{attribute 'linkalways'} 
{attribute 'no_explicit_call' := 'This FB is a CLASS and must be accessed using methods or properties'}
{attribute 'enable_dynamic_creation'}
FUNCTION_BLOCK _UDINT EXTENDS NumericDatatypeBase
VAR
	localData : UDINT;
	activeData : REFERENCE TO UDINT REF= localData;
END_VAR

PROPERTY PUBLIC Address : PVOID
GET
Address := ADR(activeData);
END_GET
END_PROPERTY

METHOD PUBLIC ClearReference
VAR_INPUT
END_VAR
activeData REF= localData;
END_METHOD

METHOD PUBLIC Clone : I_Datatype
VAR
    pClone : POINTER TO _UDINT;
END_VAR
pClone := __NEW(_UDINT(InitialValue := Value));
Clone := pClone^;
END_METHOD

METHOD FB_init : BOOL
VAR_INPUT
	bInitRetains : BOOL; // if TRUE, the retain variables are initialized (warm start / cold start)
	bInCopyCode : BOOL;  // if TRUE, the instance afterwards gets moved into the copy code (online change)
	InitialValue : UDINT;
END_VAR
localData := InitialValue;
END_METHOD

PROPERTY PUBLIC IsFloat : BOOL
GET
IsFloat := FALSE;
END_GET
END_PROPERTY

PROPERTY PUBLIC IsSigned : BOOL
GET
IsSigned := FALSE;
END_GET
END_PROPERTY

PROPERTY PUBLIC LowerBound : UDINT
GET
LowerBound := DatatypeLimits.UDINT_LOWER_LIMIT;
END_GET
END_PROPERTY

METHOD PUBLIC MakeReferenceTo
VAR_INPUT
	ReferenceTarget : REFERENCE TO UDINT;
END_VAR
activeData REF= ReferenceTarget;
END_METHOD

METHOD PROTECTED SerializeLowerbound
VAR_INPUT
	Serializer : I_Serializer;
END_VAR
Serializer.AddUdint(Lowerbound);
END_METHOD

METHOD PROTECTED SerializeUpperbound
VAR_INPUT
	Serializer : I_Serializer;
END_VAR
Serializer.AddUdint(Upperbound);
END_METHOD

METHOD PUBLIC SerializeWith
VAR_INPUT
	Serializer : I_Serializer;
END_VAR
Serializer.AddUdint(activeData);
END_METHOD

PROPERTY PUBLIC Size : UDINT
GET
Size := SIZEOF(activeData);
END_GET
END_PROPERTY

METHOD TryDeserializeFrom : BOOL
VAR_INPUT
	Deserializer : I_Deserializer;
	Feedback : I_DeserializerFeedback;
END_VAR
TryDeserializeFrom := Deserializer.TryGetUdint(activeData, Feedback);
END_METHOD

METHOD TryMakeReferenceTo : BOOL
VAR_INPUT
	Target : I_Datatype;
END_VAR
VAR
	pTargetData : POINTER TO UDINT;
END_VAR
IF NOT (Target.TypeName = TypeName) THEN
	RETURN;
END_IF

pTargetData := Target.Address;
activeData REF= pTargetData^;
TryMakeReferenceTo := TRUE;
END_METHOD

PROPERTY PUBLIC TypeName : T_MAXSTRING
GET
TypeName := 'UDINT';
END_GET
END_PROPERTY

PROPERTY PUBLIC UpperBound : UDINT
GET
UpperBound :=  DatatypeLimits.UDINT_UPPER_LIMIT;
END_GET
END_PROPERTY

PROPERTY PUBLIC Value : UDINT
GET
Value := activeData;
END_GET
SET
activeData := Value;
END_SET
END_PROPERTY

END_FUNCTION_BLOCK

(* stored: Version 1.1.0.1, ProductVersion 3.1.4024.12
   POU _UDINT: Id {71dcd266-4a01-0b15-18a9-df97eed9e923}, SpecialFunc None
   Folder Constructor: Id {b8136cbe-8219-0b2e-3211-17447d0685c4}
   Folder Protected: Id {72af1bb3-4a3e-019e-0372-5c78993bcb74}
   Property Address: Id {6b2017b6-c501-0f51-1f1c-91ce77f29f3d}
   Get Get: Id {3170fcc8-7c18-004f-1fef-c3d189cd19e7}
   Method ClearReference: Id {153f8658-897d-0f2e-0ae5-e5bf6937f727}
   Method Clone: Id {4f4b4b8f-5ab3-0d76-01cf-fcb66c7d5165}
   Method FB_init: Id {124052dd-6c04-0150-0d13-34bc3cbb9eed}
   Property IsFloat: Id {80176be4-5c58-0758-195c-1fc92db91db8}
   Get Get: Id {3a0238b2-24bc-06e9-14ab-e21bb403486a}
   Property IsSigned: Id {68e8607c-7a58-0942-36e7-b2490acbc3d7}
   Get Get: Id {2758e5f0-cda3-0ecc-2e0b-a6b9da8af3ae}
   Property LowerBound: Id {6ae77e78-4aec-07b4-3561-a3caf551a93c}
   Get Get: Id {537f398f-6575-04cc-3e14-fb4f0101f6c0}
   Method MakeReferenceTo: Id {7cc2271c-0461-003f-20e3-0c9467c7ce3a}
   Method SerializeLowerbound: Id {7468692a-27f2-0de1-1b46-f963db6307f6}
   Method SerializeUpperbound: Id {81bcf06f-dabb-0e25-1640-5c70569f4e96}
   Method SerializeWith: Id {cbc294d5-a8f9-0bd2-288a-c0159e0a6685}
   Property Size: Id {e9b4b846-21c4-08c6-2e25-7cd120957011}
   Get Get: Id {f87c64c7-3639-0bc3-1c5e-485c60388600}
   Method TryDeserializeFrom: Id {178bd17d-afcf-0727-278a-b69ee5ad5e6d}
   Method TryMakeReferenceTo: Id {796a449f-64bc-0fb8-3105-94ee489b0f37}
   Property TypeName: Id {300aba3a-3085-063b-005e-7cb8685e87e6}
   Get Get: Id {c6f8ac21-a8ee-0d6d-0d3a-019e354e5390}
   Property UpperBound: Id {b5f5f62c-c9da-077e-20d6-37607d6f5c2e}
   Get Get: Id {94193550-c19c-01b9-1aac-71fe3b85603b}
   Property Value: Id {bbe22821-5712-0854-2750-d25bafa2a285}
   Get Get: Id {1b28e4b5-db54-03be-2463-066d521080d4}
   Set Set: Id {2b3f583a-2876-0d69-1bb0-e6efed7c193b} *)
